FUNCTION F_PosZustand : STRING(80)
VAR_INPUT
	I_sString	:STRING;
	I_nStep 		:INT;
	I_sStep 		:STRING;
END_VAR
VAR
	stemp 	:STRING;
END_VAR

	stemp := 'nStep : ' (*CONCAT(I_string,' - nStep : ');*);
	stemp := CONCAT(stemp,INT_TO_STRING(I_nStep));
	stemp := CONCAT(stemp,' - ');
	stemp := CONCAT(stemp,I_sStep);


	F_PosZustand := stemp;

END_FUNCTION

(* stored: Version 1.1.0.1, ProductVersion 3.1.4024.12
   POU F_PosZustand: Id {6168bc42-9040-4099-97cf-1f776193ef61}, SpecialFunc None *)
